TYPE ST185_PnpVerPos_e :
(
    up_waiting_mover,
    down_empty,
    up_full,
    down_full,
	up_after_unload,
    _max
);
END_TYPE

(* stored: Version 1.1.0.1, ProductVersion 3.1.4024.6
   DUT ST185_PnpVerPos_e: Id {664742c8-16bc-404c-8b16-2099cc51cb79} *)
